PROGRAM prgGrid
VAR
	lrGridPower	: LREAL; //{#lynus.ag#()}
END_VAR

lrGridPower := prgEM.lrEMConsumption + prgCS.lrCSpower - prgPV.lrPVpower;

END_PROGRAM

(* stored: Version 1.1.0.1, ProductVersion 3.1.4024.11
   POU prgGrid: Id {e97f05f6-61ec-48d7-bcc3-229afa55381d}, SpecialFunc None *)
